PROGRAM Compilation
VAR
	
END_VAR

END_PROGRAM

(* stored: Version 1.1.0.1, ProductVersion 3.1.4024.15
   POU Compilation: Id {0f17c587-b026-48f1-9b9b-d704338eca71}, SpecialFunc None *)
